(* IEC 61131-3 sources: plcassist-cli/packages/volt-lsp-iec/test-corpus/lenze-mid/Device/Plc Logic/Application/A71_LocalSources/General, 8 files *)

(* ---- ATD_SR.fun ---- *)
FUNCTION ATD_SR : bool
VAR_INPUT
	iSet:BOOL;
	iReset: BOOL;
END_VAR
VAR
END_VAR
VAR_IN_OUT
	ioSR_value: BOOL;
END_VAR

ioSR_value S=iSet;
ioSR_value R=iReset;

END_FUNCTION

(* ---- fc_DintToTime.fun ---- *)
FUNCTION fc_DintToTime : time
VAR_INPUT
	DintTime: DINT;
	DecShift: DINT :=0;
END_VAR
VAR
END_VAR

fc_DintToTime:=DINT_TO_TIME(DintTime*1000/REAL_TO_DINT(EXPT(10,DecShift)));

END_FUNCTION

(* ---- RPM_To_DriveSpeed.fun ---- *)
FUNCTION RPM_To_DriveSpeed : bool
VAR_INPUT
	iEN: BOOL;
	iRPM: INT;
END_VAR
VAR
END_VAR
VAR_OUTPUT
	oDriveSpeed: INT;
END_VAR

NETWORK 0 LD
  LET en1 := ;
  IF en1 THEN oDriveSpeed := (iRPM * 6); END_IF
END_NETWORK

END_FUNCTION

(* ---- Bools_To_Byte.fb ---- *)
FUNCTION_BLOCK Bools_To_Byte
VAR
start1: POINTER TO BOOL;

i: USINT;
len: USINT;
byteval: BYTE;
END_VAR
VAR_INPUT
	adr_bit0_Of_Byte: POINTER TO bool;
END_VAR
VAR_OUTPUT
	oByte: BYTE;
END_VAR

len:=7;
oByte:=0;

start1:= adr_bit0_Of_Byte;
oByte.0:= BOOL_TO_BIT(start1^);

start1:=adr_bit0_Of_Byte+1;
oByte.1:= BOOL_TO_BIT(start1^);

start1:=adr_bit0_Of_Byte+2;
oByte.2:= BOOL_TO_BIT(start1^);

start1:=adr_bit0_Of_Byte+3;
oByte.3:= BOOL_TO_BIT(start1^);

start1:=adr_bit0_Of_Byte+4;
oByte.4:= BOOL_TO_BIT(start1^);

start1:=adr_bit0_Of_Byte+5;
oByte.5:= BOOL_TO_BIT(start1^);

start1:=adr_bit0_Of_Byte+6;
oByte.6:= BOOL_TO_BIT(start1^);

start1:=adr_bit0_Of_Byte+7;
oByte.7:= BOOL_TO_BIT(start1^);

END_FUNCTION_BLOCK

(* ---- Byte_To_Bools.fb ---- *)
FUNCTION_BLOCK Byte_To_Bools
VAR
start1: POINTER TO BOOL;

i: USINT;
len: USINT;
tempByte: BYTE;
END_VAR
VAR_INPUT
	adr_bit0_Of_Byte: POINTER TO BOOL;
END_VAR
VAR_OUTPUT
	oByte: BYTE;
END_VAR

len:=7;
oByte:=0;

start1:= adr_bit0_Of_Byte;

FOR i := 0 TO len DO
	tempByte:=REAL_TO_BYTE(EXPT(2,i));
    start1^:= BYTE_TO_BOOL((oByte AND tempByte)/tempByte);
END_FOR

END_FUNCTION_BLOCK

(* ---- GeneralMachineFlags.fb ---- *)
FUNCTION_BLOCK GeneralMachineFlags
VAR_INPUT
	iStartResetSeparate:BOOL;
	iServiceButtonHasResetFunction:BOOL;
	iFirstCycle:BOOL;
	iSignalPulse:BOOL;
	iAirPressureDoorsSeparate:BOOL;
	iEmergencyUnitOK:BOOL;
	iDoorUnitOK:BOOL;
	iSTO_Enabled:BOOL;
	iAirPressureOK:BOOL;
	iSwitchService:BOOL;
	iButtonService:BOOL;
	iStart1:BOOL;
	iStop1:BOOL;
	iReset1:BOOL;
	iAutoManual1:BOOL;
	iStart2:BOOL;
	iStop2:BOOL;
	iReset2:BOOL;
	iAutoManual2:BOOL;
	iStart3:BOOL;
	iStop3:BOOL;
	iReset3:BOOL;
	iAutoManual3:BOOL;
	iPreDelayAfterEmergStop: TIME;
	iPreStartDelayAuxDrives: TIME;
	iPreStopDelayAuxDrives: TIME;
	iPreDelayAfterSTOEnabled: TIME;

END_VAR
VAR_OUTPUT
	oResetEmergencyUnit:BOOL;
	oResetDoorUnit:BOOL;
	oStart1:BOOL;
	oStop1:BOOL;
	oReset1:BOOL;
	oCrossingDoorCircuit1:BOOL;
	oStart2:BOOL;
	oStop2:BOOL;
	oReset2:BOOL;
	oCrossingDoorCircuit2:BOOL;
	oStart3:BOOL;
	oStop3:BOOL;
	oReset3:BOOL;
	oCrossingDoorCircuit3:BOOL;
	oAlarm:BOOL;

END_VAR
VAR_IN_OUT
	GenFlags	: UDT_GeneralFlags;
END_VAR
VAR
	OneShotStart1: R_TRIG;
	OneShotStart2: R_TRIG;
	OneShotReset1: R_TRIG;
	OneShotReset2: BOOL;
	DnStartDelayAuxDrives: BOOL;
	DnStopDelayAuxDrives: BOOL;
	DnManualStopAuxDrives: BOOL;

	OffDelayPneumPressurised: TOF;
	OffDelayPneumSafetyGuard: TOF;
	OffDelayPneumEStop: TOF;

	OnDelayAfterEmergencyStop: TON;
	OnDelayStopAuxDrives: TON;
	OnDelayAfterSTOEnabled: TON;
	OnDelayManStopAuxDrives: TON;
	OnDelayStartAuxDrives: TON;

	RunAuto: SR;

END_VAR

NETWORK 0 LD TITLE: "NETWORK 2: Startup delay after emergency stop"
  GenFlags.DelayAfterEmergStop := OnDelayAfterEmergencyStop(IN := (NOT iFirstCycle AND iEmergencyUnitOK), PT := iPreDelayAfterEmergStop);
END_NETWORK
NETWORK 1 LD TITLE: "NETWORK 3: Startup delay after STO has been enabled"
  GenFlags.DelayAfterSTO := OnDelayAfterSTOEnabled(IN := (GenFlags.DelayAfterEmergStop AND iSTO_Enabled), PT := iPreDelayAfterSTOEnabled);
END_NETWORK
NETWORK 2 LD TITLE: "NETWORK 4: Stop delay auxiliary drives"
  LET g28 := (GenFlags.EnableAuxDrive AND NOT GenFlags.StartFlag AND DnStartDelayAuxDrives AND NOT GenFlags.DriveIsRunning AND NOT GenFlags.Rotflag);
  DnStopDelayAuxDrives := OnDelayStopAuxDrives(IN := g28, PT := iPreStopDelayAuxDrives);
  LET en1 := ;
  IF en1 THEN (iPreStopDelayAuxDrives = T#0MS); END_IF
  DnStopDelayAuxDrives := (g28 AND (en1 OR DnStopDelayAuxDrives));
END_NETWORK
NETWORK 3 LD TITLE: "NETWORK 5: Manual stop auxiliary drives"
  DnManualStopAuxDrives := OnDelayManStopAuxDrives(IN := (GenFlags.EnableAuxDrive AND (NOT iStop1 OR NOT iStop2 OR NOT iStop3)), PT := T#2S);
END_NETWORK
NETWORK 4 LD TITLE: "NETWORK 6: Startup delay auxiliary drives"
  LET g47 := True;
  LET g48 := (g47 AND GenFlags.EnableAuxDrive AND NOT GenFlags.AuxDrivesStarted);
  DnStartDelayAuxDrives := OnDelayStartAuxDrives(IN := g48, PT := iPreStartDelayAuxDrives);
  LET en1 := ;
  IF en1 THEN (iPreStartDelayAuxDrives = T#0MS); END_IF
  DnStartDelayAuxDrives := (g48 AND (en1 OR DnStartDelayAuxDrives));
  GenFlags.AuxDrivesStarted R= g47;
END_NETWORK
NETWORK 5 LD TITLE: "NETWORK 7: Enable markers"
  LET g190 := (GenFlags.DelayAfterEmergStop AND NOT GenFlags.MajorAlarm);
  LET g191 := (g190 AND iDoorUnitOK);
  GenFlags.EnableControl := (g191 AND NOT GenFlags.DisableControl);
  GenFlags.EnableMainDrive := (g191 AND GenFlags.EnableAuxDrive AND NOT GenFlags.AuxDrivesStarted AND DnStartDelayAuxDrives);
  GenFlags.EnableAuxDrive := (g190 AND (GenFlags.StartFlag OR (GenFlags.RunAuto AND GenFlags.RestartAuxDrives) OR (GenFlags.EnableAuxDrive AND NOT DnStopDelayAuxDrives AND NOT DnManualStopAuxDrives)));
END_NETWORK
NETWORK 6 LD TITLE: "NETWORK 8: Pneumatic markers"
  LET g118 := iEmergencyUnitOK;
  GenFlags.EnablePneumEStop := OffDelayPneumEStop(IN := g118, PT := T#1S);
  LET g119 := (g118 AND (iSTO_Enabled OR NOT iAirPressureDoorsSeparate));
  GenFlags.EnablePneumSafetyGuard := OffDelayPneumSafetyGuard(IN := g119, PT := T#1S);
  GenFlags.EnablePneumPressurised := OffDelayPneumPressurised(IN := (g119 AND iAirPressureOK), PT := T#1S);
END_NETWORK
NETWORK 7 LD TITLE: "NETWORK 9: Active control panel"
  LET g159 := True;
  GenFlags.ControlService := (g159 AND iSwitchService);
  LET g160 := (g159 AND NOT iSwitchService);
  GenFlags.ControlMan1 := (g160 AND iAutoManual1 AND NOT iAutoManual2 AND NOT iAutoManual3);
  LET g161 := (g160 AND NOT iAutoManual1);
  GenFlags.ControlMan2 := (g161 AND iAutoManual2 AND NOT iAutoManual3);
  LET g162 := (g161 AND NOT iAutoManual2);
  GenFlags.ControlMan3 := (g162 AND iAutoManual3);
  GenFlags.ControlAuto := (g162 AND NOT iAutoManual3);
END_NETWORK
NETWORK 8 LD TITLE: "NETWORK 10: Control manual"
  GenFlags.RunMan := (GenFlags.EnableControl AND ((GenFlags.ControlService AND iButtonService) OR (GenFlags.ControlMan1 AND iStart1) OR (GenFlags.ControlMan2 AND iStart2) OR (GenFlags.ControlMan3 AND iStart3)) AND iStop1 AND iStop2 AND iStop3);
END_NETWORK
NETWORK 9 LD TITLE: "NETWORK 11: Control automatic"
  GenFlags.RunAuto := RunAuto(SET1 := (GenFlags.EnableControl AND GenFlags.ControlAuto AND (iStart1 OR iStart2 OR iStart3) AND iStop1 AND iStop2 AND iStop3), RESET := (GenFlags.RunAuto AND (NOT GenFlags.EnableControl OR NOT GenFlags.ControlAuto OR NOT iStop1 OR NOT iStop2 OR NOT iStop3 OR (NOT GenFlags.DriveIsRunning AND (GenFlags.MinorAlarm OR GenFlags.MajorAlarm)))));
END_NETWORK
NETWORK 10 LD TITLE: "DONE NETWORK 12: Start pulse"
  GenFlags.StartFlag := ((OneShotStart1(CLK := ((GenFlags.ControlService AND iButtonService) OR (GenFlags.ControlMan1 AND iStart1) OR (GenFlags.ControlMan2 AND iStart2) OR (GenFlags.ControlMan3 AND iStart3) OR (GenFlags.ControlAuto AND (iStart1 OR iStart2 OR iStart3)) OR OneShotStart2.Q)) AND iStop1 AND iStop2 AND iStop3) OR OneShotStart2(CLK := (GenFlags.RunMan OR GenFlags.RunAuto)));
END_NETWORK
NETWORK 11 LD TITLE: "DONE NETWORK 13: Reset pulse"
  GenFlags.ResetFlag := ((OneShotReset1(CLK := ((GenFlags.ControlService AND ((iServiceButtonHasResetFunction AND iButtonService) OR iReset1 OR iReset2 OR iReset3)) OR ((GenFlags.ControlMan1 OR GenFlags.ControlMan2 OR GenFlags.ControlMan3 OR GenFlags.ControlAuto) AND (iReset1 OR iReset2 OR iReset3)))) AND iStop1 AND iStop2 AND iStop3) OR (NOT iStartResetSeparate AND GenFlags.StartFlag));
END_NETWORK
NETWORK 12 LD TITLE: "DONE NETWORK 14: Stop flag"
  GenFlags.StopFlag := (NOT iStop1 OR NOT iStop2 OR NOT iStop3 OR (GenFlags.StopFlag AND NOT GenFlags.StartFlag));
END_NETWORK
NETWORK 13 LD TITLE: "DONE NETWORK 15: Reset safety unit"
  oResetEmergencyUnit := ((NOT iEmergencyUnitOK OR (iEmergencyUnitOK AND NOT iDoorUnitOK)) AND ((iStartResetSeparate AND (((GenFlags.ControlMan1 OR GenFlags.ControlMan2 OR GenFlags.ControlMan3 OR GenFlags.ControlAuto) AND (iReset1 OR iReset2 OR iReset3)) OR (GenFlags.ControlService AND ((iServiceButtonHasResetFunction AND iButtonService) OR iReset1 OR iReset2 OR iReset3)))) OR (NOT iStartResetSeparate AND (((GenFlags.ControlMan1 OR GenFlags.ControlAuto) AND iStart1) OR ((GenFlags.ControlMan2 OR GenFlags.ControlAuto) AND iStart2) OR ((GenFlags.ControlMan3 OR GenFlags.ControlAuto) AND iStart3) OR (GenFlags.ControlService AND iButtonService)) AND iStop1 AND iStop2 AND iStop3)));
END_NETWORK
NETWORK 14 LD TITLE: "DONE NETWORK 16: Reset door unit"
  oResetDoorUnit := (iEmergencyUnitOK AND NOT iDoorUnitOK AND ((iStartResetSeparate AND (((GenFlags.ControlMan1 OR GenFlags.ControlMan2 OR GenFlags.ControlMan3 OR GenFlags.ControlAuto) AND (iReset1 OR iReset2 OR iReset3)) OR (GenFlags.ControlService AND ((iServiceButtonHasResetFunction AND iButtonService) OR iReset1 OR iReset2 OR iReset3)))) OR (NOT iStartResetSeparate AND (((GenFlags.ControlMan1 OR GenFlags.ControlAuto) AND iStart1) OR ((GenFlags.ControlMan2 OR GenFlags.ControlAuto) AND iStart2) OR ((GenFlags.ControlMan3 OR GenFlags.ControlAuto) AND iStart3) OR (GenFlags.ControlService AND iButtonService)) AND iStop1 AND iStop2 AND iStop3)));
END_NETWORK
NETWORK 15 LD TITLE: "DONE NETWORK 17: Crossing doorcircuit control panel 1"
  oCrossingDoorCircuit1 := GenFlags.ControlMan1;
END_NETWORK
NETWORK 16 LD TITLE: "DONE NETWORK 18: Crossing doorcircuit control panel 2"
  oCrossingDoorCircuit2 := GenFlags.ControlMan2;
END_NETWORK
NETWORK 17 LD TITLE: "DONE NETWORK 19: Crossing doorcircuit control panel 3"
  oCrossingDoorCircuit3 := GenFlags.ControlMan3;
END_NETWORK
NETWORK 18 LD TITLE: "DONE NETWORK 20: Signal lamps control panel 1"
  LET g187 := True;
  oStart1 := (g187 AND (GenFlags.ControlMan1 OR GenFlags.ControlAuto) AND (((GenFlags.RunMan OR GenFlags.RunAuto) AND NOT GenFlags.MinorAlarm AND NOT GenFlags.MajorAlarm) OR ((GenFlags.EnableControl OR (NOT iStartResetSeparate AND (GenFlags.MinorAlarm OR GenFlags.MajorAlarm))) AND iSignalPulse AND ((NOT GenFlags.MinorAlarm AND NOT GenFlags.MajorAlarm) OR NOT iStartResetSeparate))));
  oStop1 := (g187 AND iEmergencyUnitOK AND (NOT GenFlags.RunMan OR NOT GenFlags.ControlMan1) AND NOT GenFlags.RunAuto);
  oReset1 := (g187 AND (GenFlags.ControlMan1 OR GenFlags.ControlMan2 OR GenFlags.ControlMan3 OR GenFlags.ControlAuto OR GenFlags.ControlService) AND (GenFlags.MinorAlarm OR GenFlags.MajorAlarm OR NOT iDoorUnitOK) AND iSignalPulse);
END_NETWORK
NETWORK 19 LD TITLE: "DONE NETWORK 21: Signal lamps control panel 2"
  LET g186 := True;
  oStart2 := (g186 AND (GenFlags.ControlMan2 OR GenFlags.ControlAuto) AND (((GenFlags.RunMan OR GenFlags.RunAuto) AND NOT GenFlags.MinorAlarm AND NOT GenFlags.MajorAlarm) OR ((GenFlags.EnableControl OR (NOT iStartResetSeparate AND (GenFlags.MinorAlarm OR GenFlags.MajorAlarm))) AND iSignalPulse AND ((NOT GenFlags.MinorAlarm AND NOT GenFlags.MajorAlarm) OR NOT iStartResetSeparate))));
  oStop2 := (g186 AND iEmergencyUnitOK AND (NOT GenFlags.RunMan OR NOT GenFlags.ControlMan1) AND NOT GenFlags.RunAuto);
  oReset2 := (g186 AND (GenFlags.ControlMan1 OR GenFlags.ControlMan2 OR GenFlags.ControlMan3 OR GenFlags.ControlAuto OR GenFlags.ControlService) AND (GenFlags.MinorAlarm OR GenFlags.MajorAlarm OR NOT iDoorUnitOK) AND iSignalPulse);
END_NETWORK
NETWORK 20 LD TITLE: "DONE NETWORK 22: Signal lamps control panel 3"
  LET g0 := True;
  oStart3 := (g0 AND (GenFlags.ControlMan3 OR GenFlags.ControlAuto) AND (((GenFlags.RunMan OR GenFlags.RunAuto) AND NOT GenFlags.MinorAlarm AND NOT GenFlags.MajorAlarm) OR ((GenFlags.EnableControl OR (NOT iStartResetSeparate AND (GenFlags.MinorAlarm OR GenFlags.MajorAlarm))) AND iSignalPulse AND ((NOT GenFlags.MinorAlarm AND NOT GenFlags.MajorAlarm) OR NOT iStartResetSeparate))));
  oStop3 := (g0 AND iEmergencyUnitOK AND (NOT GenFlags.RunMan OR NOT GenFlags.ControlMan1) AND NOT GenFlags.RunAuto);
  oReset3 := (g0 AND (GenFlags.ControlMan1 OR GenFlags.ControlMan2 OR GenFlags.ControlMan3 OR GenFlags.ControlAuto OR GenFlags.ControlService) AND (GenFlags.MinorAlarm OR GenFlags.MajorAlarm OR NOT iDoorUnitOK) AND iSignalPulse);
END_NETWORK
NETWORK 21 LD TITLE: "TODO NETWORK 23: Signal lamp alarm"
  oAlarm := ((GenFlags.Warning OR GenFlags.MinorAlarm OR GenFlags.MajorAlarm) AND iSignalPulse);
END_NETWORK
NETWORK 22 LD TITLE: "DONE NETWORK 24: Only when during a complete CPU cycle there is no alarm, the ""Active""-alarm signals are reset"
  LET g185 := True;
  GenFlags.WarningActive := (g185 AND GenFlags.Warning);
  GenFlags.MinorAlarmActive := (g185 AND GenFlags.MinorAlarm);
  GenFlags.MajorAlarmActive := (g185 AND GenFlags.MajorAlarm);
END_NETWORK
NETWORK 23 LD TITLE: "DONE NETWORK 25: Reset alarm actions"
  LET g1 := True;
  GenFlags.Warning R= g1;
  GenFlags.MinorAlarm R= g1;
  GenFlags.MajorAlarm R= g1;
  GenFlags.DummyWarning R= g1;
  GenFlags.DisableControl R= g1;
END_NETWORK
NETWORK 24 LD TITLE: "TODO NETWORK 26: SAVE"
END_NETWORK

END_FUNCTION_BLOCK

(* ---- GeneralProgramFlags.prg ---- *)
PROGRAM GeneralProgramFlags
VAR_INPUT
END_VAR
VAR_OUTPUT
END_VAR
VAR
	AlwaysOff: BOOL;
	AlwaysOn: BOOL;
	OS: BOOL;
	first: BOOL;
	flag: BOOL;
	OSfirstflagcycle: BOOL;
	FirstCycle: BOOL;
	dummyWord: INT;
	tmr_FF500ms: TON;
	tmr_FF500ms_not: TON;
	tmr_FF100ms: TON;
	tmr_FF100ms_not: TON;
	tmr_FF50ms: TON;
	tmr_FF50ms_not: TON;
	tmr_FF1s: TON;
	tmr_FF1s_not: TON;
	PLC_StartUp_Delay: TON;
END_VAR

NETWORK 0 LD
  // Always Off
  AlwaysOff R= AlwaysOff;
END_NETWORK
NETWORK 1 LD
  // Always ON
  AlwaysOn S= NOT AlwaysOn;
END_NETWORK
NETWORK 2 LD
  FirstCycle R= (AlwaysOn AND OSfirstflagcycle);
END_NETWORK
NETWORK 3 LD
  LET en1 := AlwaysOn;
  IF en1 THEN dummyWord := MOVE(0); END_IF
END_NETWORK
NETWORK 4 LD
  LET g2 := ;
  FF50ms := tmr_FF50ms(IN := (g2 AND NOT tmr_FF50ms_not.Q), PT := T#100MS);
  LST_General.Imp100ms := tmr_FF50ms_not(IN := (g2 AND FF50ms), PT := T#100MS);
END_NETWORK
NETWORK 5 LD
  LET g1 := ;
  FF100ms := tmr_FF100ms(IN := (g1 AND NOT tmr_FF100ms_not.Q), PT := T#500MS);
  LST_General.Imp200ms := tmr_FF100ms_not(IN := (g1 AND FF100ms), PT := T#500MS);
END_NETWORK
NETWORK 6 LD
  LET g3 := ;
  FF500ms := tmr_FF500ms(IN := (g3 AND NOT tmr_FF500ms_not.Q), PT := T#500MS);
  LST_General.Imp1s := tmr_FF500ms_not(IN := (g3 AND FF500ms), PT := T#500MS);
END_NETWORK
NETWORK 7 LD
  LET g4 := ;
  FF1s := tmr_FF1s(IN := (g4 AND NOT tmr_FF1s_not.Q), PT := T#1S);
  tmr_FF1s_not(IN := (g4 AND FF1s), PT := T#1S);
END_NETWORK
NETWORK 8 LD
  LST_General.StartUpDelayPLC := PLC_StartUp_Delay(IN := AlwaysOn, PT := T#60S);
END_NETWORK

END_PROGRAM

(* ---- Simulation.prg ---- *)
PROGRAM Simulation
VAR
	ATD_Simulate: BOOL;
END_VAR

IF (ATD_Simulate) THEN
Mach1_Safety.Status.Emergency_button01:=TRUE;
Mach1_Safety.Status.Emergency_button02:=TRUE;
Mach1_Safety.Status.Emergency_button03:=TRUE;
Mach1_Safety.Status.Emergency_button04:=TRUE;
Mach1_Safety.Status.Emergency_button05:=TRUE;
Mach1_Safety.Status.EmergencyStopOK :=TRUE;

LST_InputsOutputs.I100_2_Pushbutton_stop_OP0a:=TRUE;
LST_InputsOutputs.I132_2_PB_Stop_OP2a :=TRUE;
LST_InputsOutputs.I100_0_AirpressureOK:=TRUE;
LST_InputsOutputs.I100_3_Selector_switch_auto_manual_OP0a:=FALSE;
LST_InputsOutputs.I100_1_Pushbutton_start_OP0a:=TRUE;

END_IF

END_PROGRAM
